// TIA Portal project "countingg" (V16)

(* hardware
DEVICE "HMI_1"  KTP700 Basic DP
   slot 0: "HMI_1"  KTP700 Basic DP  6AV2 123-2GA03-0AX0  16.0.0.0
   slot 1: "HMI_RT_1"  KTP700 Basic DP  6AV2 123-2GA03-0AX0  16.0.0.0
   slot 7: "HMI_1.MPI/DP_CP_1"  MPI/DP Interface  16.0.0.0
DEVICE "S7300/ET200M station_1"  S7-300 station
   slot 0: "Rail_0"  Rail  6ES7 390-1***0-0AA0
   slot 2: "PLC_1"  CPU 314C-2 DP  6ES7 314-6CH04-0AB0  V3.3
      slot 0: "MPI interface_1"  MPI
      slot 1: "DP interface_1"  DP
      slot 2: "DI 24/DO 16_1"  DI24/DO16
      slot 3: "AI 5/AO 2_1"  AI5/AO2
      slot 4: "Count_1"  Counter
      slot 5: "Positioning_1"  Positioning
*)

// ===== PLC "PLC_1"  CPU 314C-2 DP =====

VAR_GLOBAL   // PLC tag table "Default tag table"
   "Start" AT %M0.0 : Bool;
   "Stop" AT %M0.1 : Bool;
   "laser sensor" AT %M0.2 : Bool;
   "conveyer belt" AT %Q0.0 : Bool;
   "light" AT %Q0.1 : Bool;
   "counter" AT %C0 : Counter;
   "timer" AT %T0 : Timer;
   "counter output" AT %MW1 : Int;
   "reset" AT %Q0.3 : Bool;
   "restart" AT %Q0.4 : Bool;
   "output" AT %Q0.5 : Bool;
END_VAR

ORGANIZATION_BLOCK "Main"   // OB1, LAD
TITLE = "Main Program Sweep (Cycle)"
{ S7_Optimized_Access := 'FALSE' }
VERSION : 0.1
   VAR_TEMP
      OB1_EV_CLASS : Byte;   // Bits 0-3 = 1 (Coming event), Bits 4-7 = 1 (Event class 1)
      OB1_SCAN_1 : Byte;   // 1 (Cold restart scan 1 of OB 1), 3 (Scan 2-n of OB 1)
      OB1_PRIORITY : Byte;   // Priority of OB Execution
      OB1_OB_NUMBR : Byte;   // 1 (Organization block 1, OB1)
      OB1_RESERVED_1 : Byte;   // Reserved for system
      OB1_RESERVED_2 : Byte;   // Reserved for system
      OB1_PREV_CYCLE : Int;   // Cycle time of previous OB1 scan (milliseconds)
      OB1_MIN_CYCLE : Int;   // Minimum cycle time of OB1 (milliseconds)
      OB1_MAX_CYCLE : Int;   // Maximum cycle time of OB1 (milliseconds)
      OB1_DATE_TIME : Date_And_Time;   // Date and time OB1 started
      restart : Bool;
   END_VAR
   VAR_TEMP   // added for the SCL form of the ladder/FBD networks
      _w1 : Bool;
      _w2 : Bool;
      _s5time1 : S5Time;
   END_VAR
BEGIN

REGION Network 1
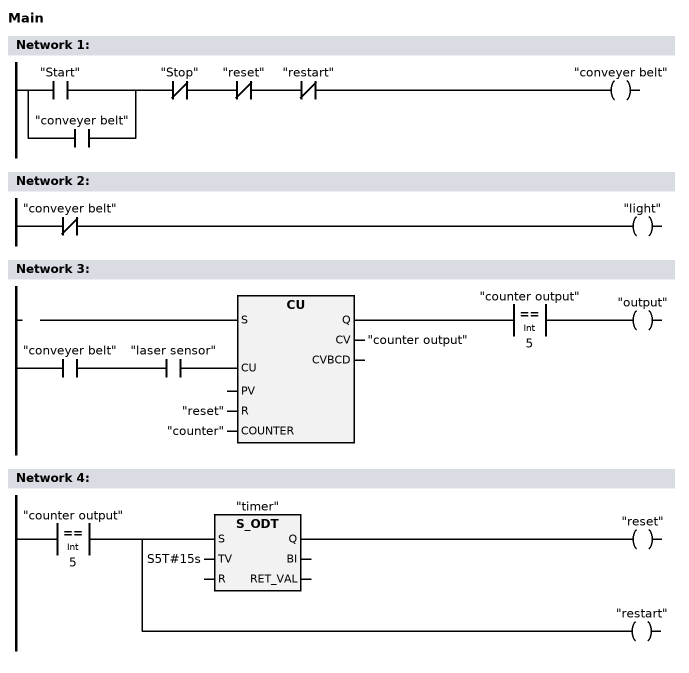
   RUNG wire#powerrail
      Contact( "Start" )
      wire#w1
      I_Contact( "Stop" )
      I_Contact( "reset" )
      I_Contact( "restart" )
      Coil( "conveyer belt" )
   END_RUNG
   RUNG wire#powerrail
      Contact( "conveyer belt" )
   END_RUNG wire#w1
   // the same network as SCL:
   "conveyer belt" := ("Start" OR "conveyer belt") AND NOT "Stop" AND NOT "reset" AND NOT "restart";
END_REGION

REGION Network 2
   RUNG wire#powerrail
      I_Contact( "conveyer belt" )
      Coil( "light" )
   END_RUNG
   // the same network as SCL:
   "light" := NOT "conveyer belt";
END_REGION

REGION Network 3
   // no SCL statement known for Cu: written as a call
   Cu(cu := "conveyer belt" AND "laser sensor",
      r := "reset",
      "counter" := "counter",
      q => #_w1,
      cv => "counter output");
   "output" := #_w1 AND ("counter output" = 5);
END_REGION

REGION Network 4
   RUNG wire#powerrail
      { S7_Templates := "SrcType := Int" } EQ_Contact(in1 := "counter output", in2 := 5)
      wire#w1
      S_ODT(T_NO := "timer", TV := S5T#15s, R :=, BI =>, RET_VAL =>)
      Coil( "reset" )
   END_RUNG
   RUNG wire#w1
      Coil( "restart" )
   END_RUNG
   // the same network as SCL:
   #_w1 := "counter output" = 5;
   #_s5time1 := S_ODT(T_NO := "timer", S := #_w1, TV := S5T#15s, Q => #_w2);
   "reset" := #_w2;
   "restart" := #_w1;
END_REGION
END_ORGANIZATION_BLOCK

(* ===== HMI "HMI_RT_1" =====
system functions are stored by id; their names below are inferred from use
connection "HMI_Connection_1": IF1 B, SIMATIC S7 300/400 MPI

HMI tags "Default tag table"
   "Tag_ScreenNumber" : UInt, internal
   "light" : Bool = PLC light AT %Q0.1, 1 s
   "laser sensor" : Bool = PLC "laser sensor" AT %M0.2, 1 s
   "Start" : Bool = PLC Start AT %M0.0, 1 s
   "Stop" : Bool = PLC Stop AT %M0.1, 1 s
   "counter output" : Int = PLC "counter output" AT %MW1, 1 s
   "Move" : Int, internal
   "output" : Bool = PLC output AT %Q0.5, 1 s
   "conveyer belt" : Bool = PLC "conveyer belt" AT %Q0.0, 1 s

Template "Template_1" 800x480
   Button "Exit" at 714,429 size 71x50; TextOff 'Exit'; PictureOff "ExitRuntime_KTP700_Basic_DP_TR"; PictureOn "ExitRuntime_KTP700_Basic_DP_TR"
      on Release: StopRuntime(0)
   Button "Template_Button" at 614,429 size 71x50; TextOff 'Text'
   Button "Template_Button_1" at 514,429 size 71x50; TextOff 'Text'
   Button "Template_Button_2" at 414,429 size 71x50; TextOff 'Text'
   Button "Template_Button_3" at 314,429 size 71x50; TextOff 'Text'
   Button "Template_Button_4" at 214,429 size 71x50; TextOff 'Text'
   Button "Alarms" at 114,429 size 71x50; TextOff 'Alarms'; PictureOff "AlarmDisplay_KTP700_Basic_DP_TR"; PictureOn "AlarmDisplay_KTP700_Basic_DP_TR"
      on Release: function_ef3f5d25("Alarm window_Unacknowledged", -1)
   Button "Start screen" at 14,429 size 71x50; TextOff 'Start screen'; PictureOff "NavigateHome_KTP700_Basic_DP_TR"; PictureOn "NavigateHome_KTP700_Basic_DP_TR"
      on Release: ActivateScreen("Root screen", 0)
   SymbolicIOField "Symbolic_IO_Field_Screen" at 93,9 size 600x33; TextOff '0'; TextOn '1'; TextList "TextList_ScreenNames"
      ProcessValue <- "Tag_ScreenNumber"
      on Change: ActivateScreenByNumber("Tag_ScreenNumber", 0)
   DateTimeField "HmiScreenItemData" at 695,25 size 105x25
   DateTimeField "HmiScreenItemData_1" at 695,0 size 105x25
   GraphicView "Logo" at 0,0 size 91x51; Picture "Logo of HMI_1"

screen "Root screen" 800x480, template "Template_1"
   on GenerateScreen: SetTag("Tag_ScreenNumber", 1); function_f9c01323("Move", 1, 100, 0, 1)
   Circle "Circle_1" at 646,61 size 78x78
      Appearance <- "light"
   Button "Button_1" at 44,61 size 96x32; TextOff 'Start'
      on Press: SetBit("Start")
      on Release: ResetBit("Start")
   Button "Button_2" at 42,124 size 96x32; TextOff 'Stop'
      on Release: ResetBit("Stop")
      on Press: SetBit("Stop")
   Button "Button_3" at 479,77 size 96x32; TextOff 'Counter'
      on Press: SetBit("laser sensor")
      on Release: ResetBit("laser sensor")
   GraphicView "Graphic view_1" at 76,307 size 400x58; Picture "Graphic_1"
   GraphicView "Graphic view_2" at 80,357 size 126x64; Picture "Graphic_2"
   GraphicView "Graphic view_3" at 130,247 size 48x87; Picture "Graphic_3"
      HorizontalMovement <- "Move"
      Visibility <- "conveyer belt"
   GraphicView "Graphic view_4" at 381,157 size 41x77; Picture "Graphic_4"
   GraphicView "Graphic view_6" at 118,249 size 48x87; Picture "Graphic_3"
   IOField "I/O field_1" at 485,124 size 96x32; FormatPattern s99999
      ProcessValue <- "counter output"
*)